// TIA Portal V21 export
TYPE "Dane"
   STRUCT
      z1 : Bool;
      z2 : Bool;
      "string" : String;
   END_STRUCT;
END_TYPE
